FUNCTION_BLOCK PUBLIC FB_PalletStop EXTENDS FB_IndexedPosition

VAR_IN_OUT
	HardwareInputArray 	: ARRAY [*] OF BOOL;		// For Actuators
	//Upstream			: DWORD;
	//Downstream			: DWORD;
END_VAR

VAR
	Configuration 			: ST_PalletStopConfiguration;
	Status					: ST_PalletStopStatus;
	InitDone 				: BOOL := FALSE;
	PalletStopHardwareState	: DINT := E_PalletStopHardwareStates.Lowered;
END_VAR

IF NOT InitDone THEN
	M_Init();
	InitDone:= TRUE;
ELSE
	SUPER^();
	M_Cyclic();
	M_StateMachine();
END_IF

METHOD PRIVATE M_Cyclic : BOOL
VAR_INPUT
END_VAR
Controls.isDefined := TRUE; // I exist
Configuration.DownstreamOutputArrayPosition 	:= Configuration.DownstreamHardwareOutput - 32768;
HardwareInputArray[Configuration.DownstreamOutputArrayPosition] 	:= SEL( PalletStopHardwareState = E_PalletStopHardwareStates.Raised OR PalletStopHardwareState = E_PalletStopHardwareStates.Raising, FALSE, TRUE);
END_METHOD

METHOD PRIVATE M_Init : BOOL
VAR_INPUT
END_VAR
END_METHOD

METHOD PUBLIC M_Reset : BOOL
VAR_INPUT
END_VAR
PalletStopHardwareState := E_PalletStopHardwareStates.Lowered;

SUPER^.P_Controls.Front.Request := E_IndexedPositionSimplifiedRequest.NoRequest;
SUPER^.P_Controls.Rear.Request := E_IndexedPositionSimplifiedRequest.NoRequest;
SUPER^.P_Controls.Left.Request := E_IndexedPositionSimplifiedRequest.NoRequest;
SUPER^.P_Controls.Right.Request := E_IndexedPositionSimplifiedRequest.NoRequest;

SUPER^.P_Controls.Request := E_IndexedPositionTransitionRequest.NoRequest;
SUPER^.P_Controls.State := E_IndexedPositionStates.Starved;
END_METHOD

METHOD PRIVATE M_StateMachine : BOOL
VAR_INPUT
END_VAR
(*IF Configuration.BypassLTU THEN
	State := E_LTUStates.Bypass;
ELSE
	State := E_LTUStates.Idle;
END_IF*)
IF SUPER^.P_Controls.OperationMode THEN
	CASE SUPER^.Controls.State OF 
	// Would be better as a raise and lower requestr, followed by sensor confirmation that the Pallet Stop was raised or lowered, but no feedback from the simulation :(
		E_IndexedPositionStates.ReceivingFromRear, E_IndexedPositionStates.Idle:
			PalletStopHardwareState := E_PalletStopHardwareStates.Raised;
			
		E_IndexedPositionStates.SendingToFront, E_IndexedPositionStates.Starved:
			PalletStopHardwareState := E_PalletStopHardwareStates.Lowered;
	END_CASE
ELSE
	//
END_IF
END_METHOD

PROPERTY PUBLIC P_Configuration : REFERENCE TO ST_PalletStopConfiguration
GET
P_Configuration REF= Configuration;
END_GET
END_PROPERTY

PROPERTY PUBLIC P_Status : REFERENCE TO ST_PalletStopStatus
GET
P_Status REF= Status;
END_GET
END_PROPERTY

END_FUNCTION_BLOCK

(* stored: Version 1.1.0.1, ProductVersion 3.1.4024.12
   POU FB_PalletStop: Id {cd29b529-bf00-4cf7-b53d-66826a23232d}, SpecialFunc None
   Method M_Cyclic: Id {40493c72-3c09-41b8-996c-78bd5f629286}
   Method M_Init: Id {6260de79-2222-47bf-8a95-b48de7f82031}
   Method M_Reset: Id {c012534f-867f-417e-b453-772258b520a0}
   Method M_StateMachine: Id {411c2fb1-1cb8-41e6-97da-553355b7df91}
   Property P_Configuration: Id {83c6bb9f-3150-4335-b964-a41cdeea8c04}
   Get Get: Id {73ed7111-15eb-4947-acb8-898e68a1132e}
   Property P_Status: Id {0fc86d92-1a94-4d0f-a8f5-cdba67e8235e}
   Get Get: Id {f8cfadbb-9df5-44e6-95cb-3b56b49ed259} *)
